PROGRAM BeamEnableChain
VAR
	BeamEn	AT %Q*:BOOL;
END_VAR

BeamEn := TRUE;

END_PROGRAM

(* stored: Version 1.1.0.1, ProductVersion 3.1.4022.10
   POU BeamEnableChain: Id {09e8a53f-5084-40ca-a5ec-b6c4ff87b1a6}, SpecialFunc None *)
